# EPICS substitutions: ek9000App/Db/EL1722.substitutions
file EL1722.template
{ 	pattern
	{
		TERMINAL,

	}
	{
	}
}
